# B&R Automation Studio project GUID_Presentation
Automation Studio 4.12.1.151

## Configuration Example

CPU X20CP1586, AutomationRuntime G4.93, Build 4.1.2, Vc V4.72.6

### Task classes (Cpu.sw)
```
Cyclic#4:
  Program <- Program.prg
Libraries: Operations
```

### Hardware
```
X20CP1586 : X20CP1586 v1.10.0.0
  Connector IF2:
    ActivateDevice = 1
  ConfigurationID = GUID_Presentation_Example
  FileDevice1
  FileDeviceName1 = USER
  FileDevicePath1 = USER_PATH
```

## Logical view

Binary libraries used (declarations not repeated): operator, runtime, astime, AsIecCon, Library

### Library Logical/Libraries/Operations (IEC)

#### Types.typ - Exported data types
```iecst
TYPE
	ResultsType : 	STRUCT
		add : DINT;
		sub : DINT;
		mult : DINT;
		div : REAL;
	END_STRUCT;
END_TYPE
```

#### Operations.fun - Exported functions and function blocks
```iecst
FUNCTION Operaciones : USINT
	VAR_INPUT
		a : USINT;
		b : USINT;
		pResults : REFERENCE TO ResultsType;
	END_VAR
END_FUNCTION
```

#### Operations.st
```iecst
FUNCTION Operaciones
	pResults.add := a + b;
	pResults.sub := a - b;
	pResults.mult := a * b;
	pResults.div := a / b;
END_FUNCTION
```

### Program Logical/Program

#### Variables.var
```iecst
VAR
	Numero_A : USINT := 20;
	Numero_B : USINT := 2;
	Resultados : ResultsType;
	Contador1 : USINT := 0;
END_VAR
```

#### Main.st
```iecst
PROGRAM _INIT
	(* Insert code here *)

	Resultados;

END_PROGRAM

PROGRAM _CYCLIC
	// Release 1.0
	Operaciones( a := Numero_A,b := Numero_B,pResults := ADR(Resultados));
	counter := counter + 4;//Version mejorada final final
END_PROGRAM

PROGRAM _EXIT
	(* Insert code here *)

END_PROGRAM
```

Listed in the project but not available here: Logical/Libraries/Operations/Constants.var
